{attribute 'pack_mode' := '2'}
TYPE ST_Ctrl_NciMFuncCycle :
STRUCT
  FastMFuncMask   : ARRAY [1..5] OF DWORD;
  HskMFuncNo      : UINT;
  HskMFuncReq     : WORD;
  HFuncValue      : UDINT; 
END_STRUCT
END_TYPE

(* stored: Version 1.1.0.1, ProductVersion 3.1.4024.9
   DUT ST_Ctrl_NciMFuncCycle: Id {18e084f8-e064-0a69-2a01-ad59ea09153e} *)
